INTERFACE I_Foo

METHOD DoSomething : BOOL
VAR_INPUT
END_VAR
END_METHOD

END_INTERFACE

(* stored: Version 1.1.0.1, ProductVersion 3.1.4020.6
   Itf I_Foo: Id {cfc3bfb3-5c67-43b4-948b-3a3be13cbcab}
   Method DoSomething: Id {c723349e-b80d-4b1f-8264-307deb935307} *)
